TYPE ST_BaseControlElement_Power :
STRUCT
	cmdTurnOn				: FB_BaseCommand;
	cmdTurnOff				: FB_BaseCommand;
	bStatus					: BOOL;
END_STRUCT
END_TYPE

(* stored: Version 1.1.0.1
   DUT ST_BaseControlElement_Power: Id {53f646f7-0142-0b0d-27cd-8402c7fe716e} *)
